{attribute 'qualified_only'}
{attribute 'strict'}
TYPE eTcoUrRoboticsSimpleTests : 
(
    Restore := 1,
    CleanUp,
    Message,
    PowerDisable,
    PowerEnable,
    Reset,
    Last
);
END_TYPE

(* stored: Version 1.1.0.1, ProductVersion 3.1.4024.12
   DUT eTcoUrRoboticsSimpleTests: Id {c1207581-4710-0499-1215-86964475da8b} *)
